Staubli VAL3: checkColValue.pgx

program checkColValue(string x_sColValue, bool& x_bIsOK[])
begin
  //? asc(x_sColValue,0)
  x_bIsOK=(asc(x_sColValue,0)>=asc("a",0)) and (asc(x_sColValue,0)<=asc("z",0))
  x_bIsOK=x_bIsOK or (asc(x_sColValue,0)>=asc("A",0)) and (asc(x_sColValue,0)<=asc("Z",0))
end
